PROGRAM P_GetTime
VAR
	fbGetLocalTime  : NT_GetTime;
    bBusy           : BOOL;
    bError          : BOOL;
    nErrID          : UDINT;
    presetTime      : TIMESTRUCT;

    syncTimer       : TON;
    syncTrigger     : F_TRIG;
    bSynchronize    : BOOL;    
    
    fbRTC           : RTC;
    bValid_RTC      : BOOL;
    time_RTC        : DT;
END_VAR

syncTimer(IN:= NOT syncTimer.Q, PT:= T#500MS);

fbGetLocalTime(START:=syncTimer.Q,NETID:='',TMOUT:=T#500MS, TIMESTR => presetTime);

syncTrigger(CLK := fbGetLocalTime.BUSY AND NOT fbGetLocalTime.ERR, Q => bSynchronize);

fbRTC(EN := bSynchronize, PDT := SYSTEMTIME_TO_DT(TIMESTR:= presetTime), Q => bValid_RTC, CDT => time_RTC);

END_PROGRAM

(* stored: Version 1.1.0.1, ProductVersion 3.1.4024.3
   POU P_GetTime: Id {8bbcaad1-ef8e-49a9-8c3f-cd31343b3a7d}, SpecialFunc None *)
